FUNCTION_BLOCK DDB_EH_TimeOutComplete (* Composite FB wrapping other FBs *)
  (* Standard: 61499-2 *)
  (* Version 1.0, 2021-03-10, dummy *)
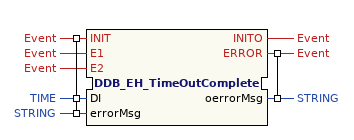
  EVENT_INPUT
    INIT WITH DI, errorMsg; (* Initialization Request *)
    E1; (* Normal Execution Request *)
    E2;
  END_EVENT
  EVENT_OUTPUT
    INITO; (* Initialization Confirm *)
    ERROR WITH oerrorMsg; (* Execution Confirmation *)
  END_EVENT
  VAR_INPUT
    DI : TIME; (* Input event qualifier *)
    errorMsg : STRING;
  END_VAR
  VAR_OUTPUT
    oerrorMsg : STRING;
  END_VAR
  FBS
    DDB_EH_TimeOut : DDB_EH_TimeOut;
    E_TimeOut : E_TimeOut;
  END_FBS
  EVENT_CONNECTIONS
    DDB_EH_TimeOut.INITO TO INITO;
    INIT TO DDB_EH_TimeOut.INIT;
    E1 TO DDB_EH_TimeOut.EI1;
    E2 TO DDB_EH_TimeOut.EI2;
    DDB_EH_TimeOut.ERROR TO ERROR;
  END_CONNECTIONS
  DATA_CONNECTIONS
    DI TO DDB_EH_TimeOut.DI1;
    errorMsg TO oerrorMsg;
  END_CONNECTIONS
  ADAPTER_CONNECTIONS
    DDB_EH_TimeOut.TimeOut TO E_TimeOut.TimeOutSocket;
  END_CONNECTIONS
END_FUNCTION_BLOCK
